# EPICS substitutions: epics/apps/caenHvApp/Db/ltcc1.substitutions
# Structure of the HV For the Low Threshold Cerenkov Counter(Abbr:LTCC)
# Geographical:
#
# HV (Abbr: HV)
#	 Slot (Abbr: Sl)
#		 Channel (Abbr: Ch)

#Detector based:
# Sector (Abbr: Sec)
# 	Side L or R (Abbr: )
# 		Element 1-18 (Abbr: )

file "db/b_templates.db" {
	pattern {Cr,	CrName,	Sl,	Ch,	Sys,	Det,	Element,    CScode, pwonoff, v0set, i0set, trip, rampup, rampdn, svmax}
		{"4",	"HVECAL1",	"14",	"0",	"HV",	"LTCC",	"Sec1_L01",	"#C3588", "S2816", "S512", "S1280", "S2560", "S1024", "S768", "S3328"}
		{"4",	"HVECAL1",	"14",	"1",	"HV",	"LTCC",	"Sec1_L02",	"#C3588", "S2817", "S513", "S1281", "S2561", "S1025", "S769", "S3329"}
		{"4",	"HVECAL1",	"14",	"2",	"HV",	"LTCC",	"Sec1_L03",	"#C3588", "S2818", "S514", "S1282", "S2562", "S1026", "S770", "S3330"}
		{"4",	"HVECAL1",	"14",	"3",	"HV",	"LTCC",	"Sec1_L04",	"#C3588", "S2819", "S515", "S1283", "S2563", "S1027", "S771", "S3331"}
		{"4",	"HVECAL1",	"14",	"4",	"HV",	"LTCC",	"Sec1_L05",	"#C3588", "S2820", "S516", "S1284", "S2564", "S1028", "S772", "S3332"}
		{"4",	"HVECAL1",	"14",	"5",	"HV",	"LTCC",	"Sec1_L06",	"#C3588", "S2821", "S517", "S1285", "S2565", "S1029", "S773", "S3333"}
		{"4",	"HVECAL1",	"14",	"6",	"HV",	"LTCC",	"Sec1_L07",	"#C3588", "S2822", "S518", "S1286", "S2566", "S1030", "S774", "S3334"}
		{"4",	"HVECAL1",	"14",	"7",	"HV",	"LTCC",	"Sec1_L08",	"#C3588", "S2823", "S519", "S1287", "S2567", "S1031", "S775", "S3335"}
		{"4",	"HVECAL1",	"14",	"8",	"HV",	"LTCC",	"Sec1_L09",	"#C3588", "S2824", "S520", "S1288", "S2568", "S1032", "S776", "S3336"}
		{"4",	"HVECAL1",	"14",	"9",	"HV",	"LTCC",	"Sec1_L10",	"#C3588", "S2825", "S521", "S1289", "S2569", "S1033", "S777", "S3337"}
		{"4",	"HVECAL1",	"14",	"10",	"HV",	"LTCC",	"Sec1_L11",	"#C3588", "S2826", "S522", "S1290", "S2570", "S1034", "S778", "S3338"}
		{"4",	"HVECAL1",	"14",	"11",	"HV",	"LTCC",	"Sec1_L12",	"#C3588", "S2827", "S523", "S1291", "S2571", "S1035", "S779", "S3339"}
		{"4",	"HVECAL1",	"14",	"12",	"HV",	"LTCC",	"Sec1_L13",	"#C3588", "S2828", "S524", "S1292", "S2572", "S1036", "S780", "S3340"}
		{"4",	"HVECAL1",	"14",	"13",	"HV",	"LTCC",	"Sec1_L14",	"#C3588", "S2829", "S525", "S1293", "S2573", "S1037", "S781", "S3341"}
		{"4",	"HVECAL1",	"14",	"14",	"HV",	"LTCC",	"Sec1_L15",	"#C3588", "S2830", "S526", "S1294", "S2574", "S1038", "S782", "S3342"}
		{"4",	"HVECAL1",	"14",	"15",	"HV",	"LTCC",	"Sec1_L16",	"#C3588", "S2831", "S527", "S1295", "S2575", "S1039", "S783", "S3343"}
		{"4",	"HVECAL1",	"14",	"16",	"HV",	"LTCC",	"Sec1_L17",	"#C3588", "S2832", "S528", "S1296", "S2576", "S1040", "S784", "S3344"}
		{"4",	"HVECAL1",	"14",	"17",	"HV",	"LTCC",	"Sec1_L18",	"#C3588", "S2833", "S529", "S1297", "S2577", "S1041", "S785", "S3345"}

		{"4",	"HVECAL1",	"15",	"0",	"HV",	"LTCC",	"Sec1_R01",	"#C3844", "S2816", "S512", "S1280", "S2560", "S1024", "S768", "S3328"}
		{"4",	"HVECAL1",	"15",	"1",	"HV",	"LTCC",	"Sec1_R02",	"#C3844", "S2817", "S513", "S1281", "S2561", "S1025", "S769", "S3329"}
		{"4",	"HVECAL1",	"15",	"2",	"HV",	"LTCC",	"Sec1_R03",	"#C3844", "S2818", "S514", "S1282", "S2562", "S1026", "S770", "S3330"}
		{"4",	"HVECAL1",	"15",	"3",	"HV",	"LTCC",	"Sec1_R04",	"#C3844", "S2819", "S515", "S1283", "S2563", "S1027", "S771", "S3331"}
		{"4",	"HVECAL1",	"15",	"4",	"HV",	"LTCC",	"Sec1_R05",	"#C3844", "S2820", "S516", "S1284", "S2564", "S1028", "S772", "S3332"}
		{"4",	"HVECAL1",	"15",	"5",	"HV",	"LTCC",	"Sec1_R06",	"#C3844", "S2821", "S517", "S1285", "S2565", "S1029", "S773", "S3333"}
		{"4",	"HVECAL1",	"15",	"6",	"HV",	"LTCC",	"Sec1_R07",	"#C3844", "S2822", "S518", "S1286", "S2566", "S1030", "S774", "S3334"}
		{"4",	"HVECAL1",	"15",	"7",	"HV",	"LTCC",	"Sec1_R08",	"#C3844", "S2823", "S519", "S1287", "S2567", "S1031", "S775", "S3335"}
		{"4",	"HVECAL1",	"15",	"8",	"HV",	"LTCC",	"Sec1_R09",	"#C3844", "S2824", "S520", "S1288", "S2568", "S1032", "S776", "S3336"}
		{"4",	"HVECAL1",	"15",	"9",	"HV",	"LTCC",	"Sec1_R10",	"#C3844", "S2825", "S521", "S1289", "S2569", "S1033", "S777", "S3337"}
		{"4",	"HVECAL1",	"15",	"10",	"HV",	"LTCC",	"Sec1_R11",	"#C3844", "S2826", "S522", "S1290", "S2570", "S1034", "S778", "S3338"}
		{"4",	"HVECAL1",	"15",	"11",	"HV",	"LTCC",	"Sec1_R12",	"#C3844", "S2827", "S523", "S1291", "S2571", "S1035", "S779", "S3339"}
		{"4",	"HVECAL1",	"15",	"12",	"HV",	"LTCC",	"Sec1_R13",	"#C3844", "S2828", "S524", "S1292", "S2572", "S1036", "S780", "S3340"}
		{"4",	"HVECAL1",	"15",	"13",	"HV",	"LTCC",	"Sec1_R14",	"#C3844", "S2829", "S525", "S1293", "S2573", "S1037", "S781", "S3341"}
		{"4",	"HVECAL1",	"15",	"14",	"HV",	"LTCC",	"Sec1_R15",	"#C3844", "S2830", "S526", "S1294", "S2574", "S1038", "S782", "S3342"}
		{"4",	"HVECAL1",	"15",	"15",	"HV",	"LTCC",	"Sec1_R16",	"#C3844", "S2831", "S527", "S1295", "S2575", "S1039", "S783", "S3343"}
		{"4",	"HVECAL1",	"15",	"16",	"HV",	"LTCC",	"Sec1_R17",	"#C3844", "S2832", "S528", "S1296", "S2576", "S1040", "S784", "S3344"}
		{"4",	"HVECAL1",	"15",	"17",	"HV",	"LTCC",	"Sec1_R18",	"#C3844", "S2833", "S529", "S1297", "S2577", "S1041", "S785", "S3345"}

}
